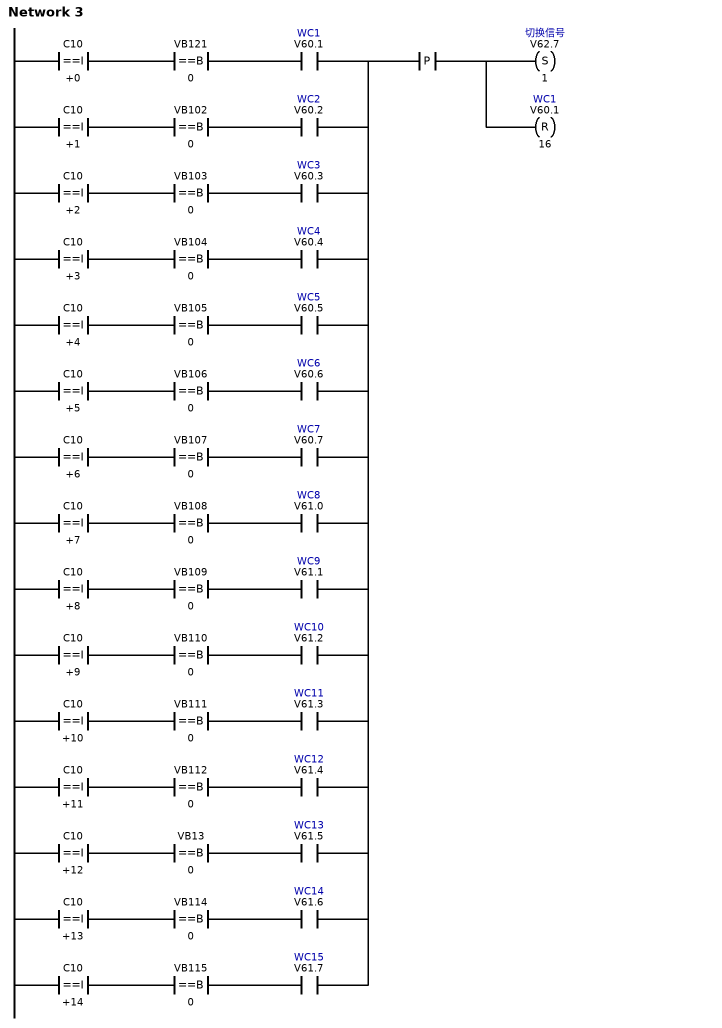
[picture p120: SBR53 networks 3-3]
Network 3
LDW=   C10, +0
AB=    VB121, 0
A      WC1:V60.1
LDW=   C10, +1
AB=    VB102, 0
A      WC2:V60.2
OLD
LDW=   C10, +2
AB=    VB103, 0
A      WC3:V60.3
OLD
LDW=   C10, +3
AB=    VB104, 0
A      WC4:V60.4
OLD
LDW=   C10, +4
AB=    VB105, 0
A      WC5:V60.5
OLD
LDW=   C10, +5
AB=    VB106, 0
A      WC6:V60.6
OLD
LDW=   C10, +6
AB=    VB107, 0
A      WC7:V60.7
OLD
LDW=   C10, +7
AB=    VB108, 0
A      WC8:V61.0
OLD
LDW=   C10, +8
AB=    VB109, 0
A      WC9:V61.1
OLD
LDW=   C10, +9
AB=    VB110, 0
A      WC10:V61.2
OLD
LDW=   C10, +10
AB=    VB111, 0
A      WC11:V61.3
OLD
LDW=   C10, +11
AB=    VB112, 0
A      WC12:V61.4
OLD
LDW=   C10, +12
AB=    VB13, 0
A      WC13:V61.5
OLD
LDW=   C10, +13
AB=    VB114, 0
A      WC14:V61.6
OLD
LDW=   C10, +14
AB=    VB115, 0
A      WC15:V61.7
OLD
EU
S      切换信号:V62.7, 1
R      WC1:V60.1, 16
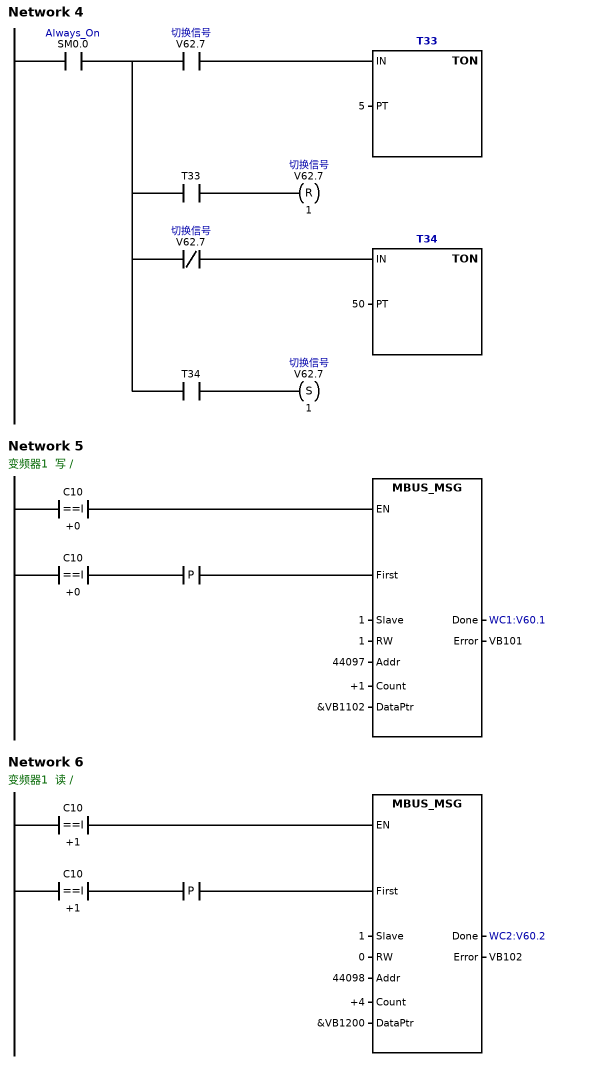
Network 4
LD     Always_On:SM0.0
LPS
A      切换信号:V62.7
TON    T33, 5
LRD
A      T33
R      切换信号:V62.7, 1
LRD
AN     切换信号:V62.7
TON    T34, 50
LPP
A      T34
S      切换信号:V62.7, 1
Network 5
// 变频器1  写
// 
LDW=   C10, +0
=      L60.0
LDW=   C10, +0
EU
=      L63.7
LD     L60.0
CALL   MBUS_MSG:SBR3, L63.7, 1, 1, 44097, +1, &VB1102, WC1:V60.1, VB101
Network 6
// 变频器1  读
// 
LDW=   C10, +1
=      L60.0
LDW=   C10, +1
EU
=      L63.7
LD     L60.0
CALL   MBUS_MSG:SBR3, L63.7, 1, 0, 44098, +4, &VB1200, WC2:V60.2, VB102
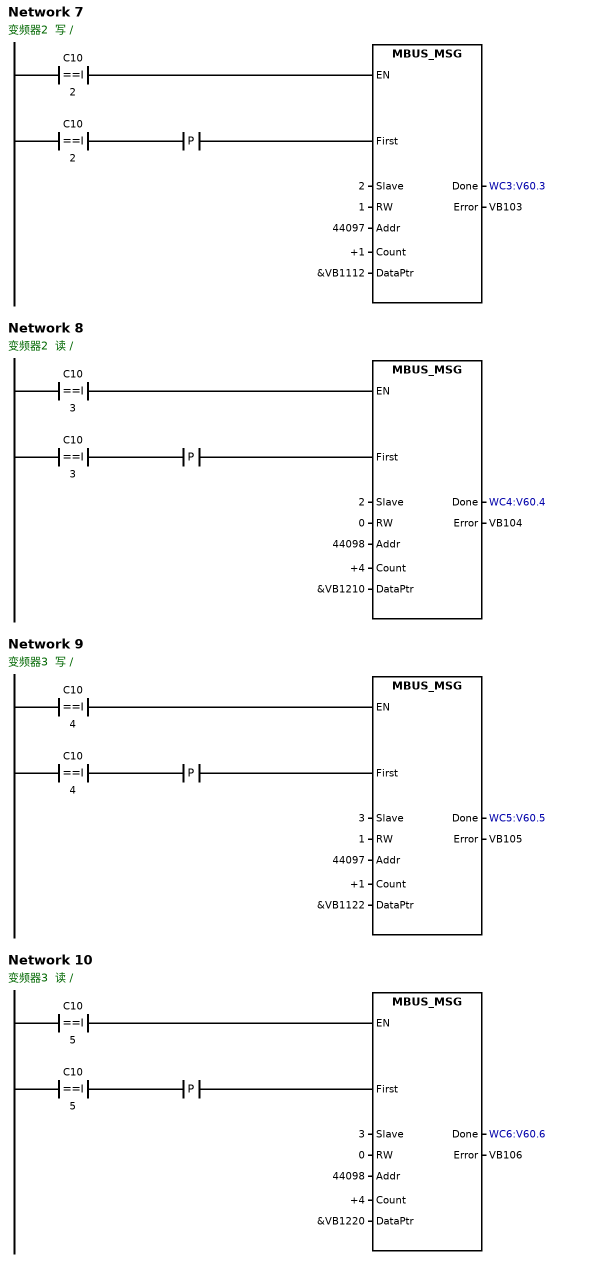
Network 7
// 变频器2  写
// 
LDW=   C10, 2
=      L60.0
LDW=   C10, 2
EU
=      L63.7
LD     L60.0
CALL   MBUS_MSG:SBR3, L63.7, 2, 1, 44097, +1, &VB1112, WC3:V60.3, VB103
Network 8
// 变频器2  读
// 
LDW=   C10, 3
=      L60.0
LDW=   C10, 3
EU
=      L63.7
LD     L60.0
CALL   MBUS_MSG:SBR3, L63.7, 2, 0, 44098, +4, &VB1210, WC4:V60.4, VB104
Network 9
// 变频器3  写
// 
LDW=   C10, 4
=      L60.0
LDW=   C10, 4
EU
=      L63.7
LD     L60.0
CALL   MBUS_MSG:SBR3, L63.7, 3, 1, 44097, +1, &VB1122, WC5:V60.5, VB105
Network 10
// 变频器3  读
// 
LDW=   C10, 5
=      L60.0
LDW=   C10, 5
EU
=      L63.7
LD     L60.0
CALL   MBUS_MSG:SBR3, L63.7, 3, 0, 44098, +4, &VB1220, WC6:V60.6, VB106
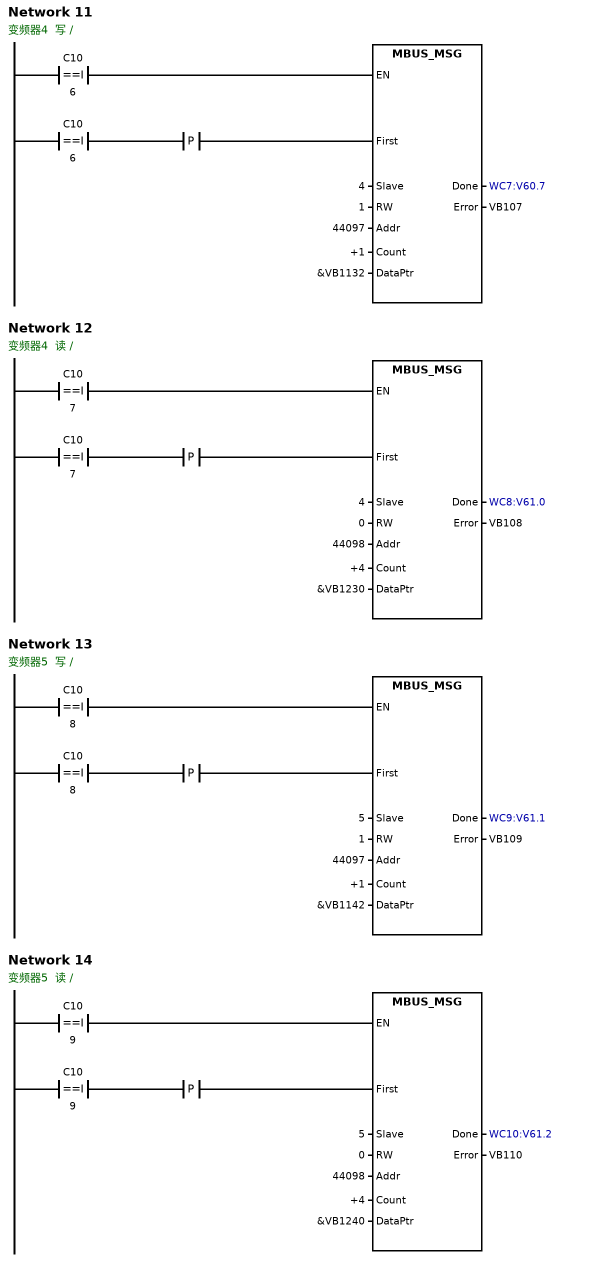
Network 11
// 变频器4  写
// 
LDW=   C10, 6
=      L60.0
LDW=   C10, 6
EU
=      L63.7
LD     L60.0
CALL   MBUS_MSG:SBR3, L63.7, 4, 1, 44097, +1, &VB1132, WC7:V60.7, VB107
Network 12
// 变频器4  读
// 
LDW=   C10, 7
=      L60.0
LDW=   C10, 7
EU
=      L63.7
LD     L60.0
CALL   MBUS_MSG:SBR3, L63.7, 4, 0, 44098, +4, &VB1230, WC8:V61.0, VB108
Network 13
// 变频器5  写
// 
LDW=   C10, 8
=      L60.0
LDW=   C10, 8
EU
=      L63.7
LD     L60.0
CALL   MBUS_MSG:SBR3, L63.7, 5, 1, 44097, +1, &VB1142, WC9:V61.1, VB109
Network 14
// 变频器5  读
// 
LDW=   C10, 9
=      L60.0
LDW=   C10, 9
EU
=      L63.7
LD     L60.0
CALL   MBUS_MSG:SBR3, L63.7, 5, 0, 44098, +4, &VB1240, WC10:V61.2, VB110
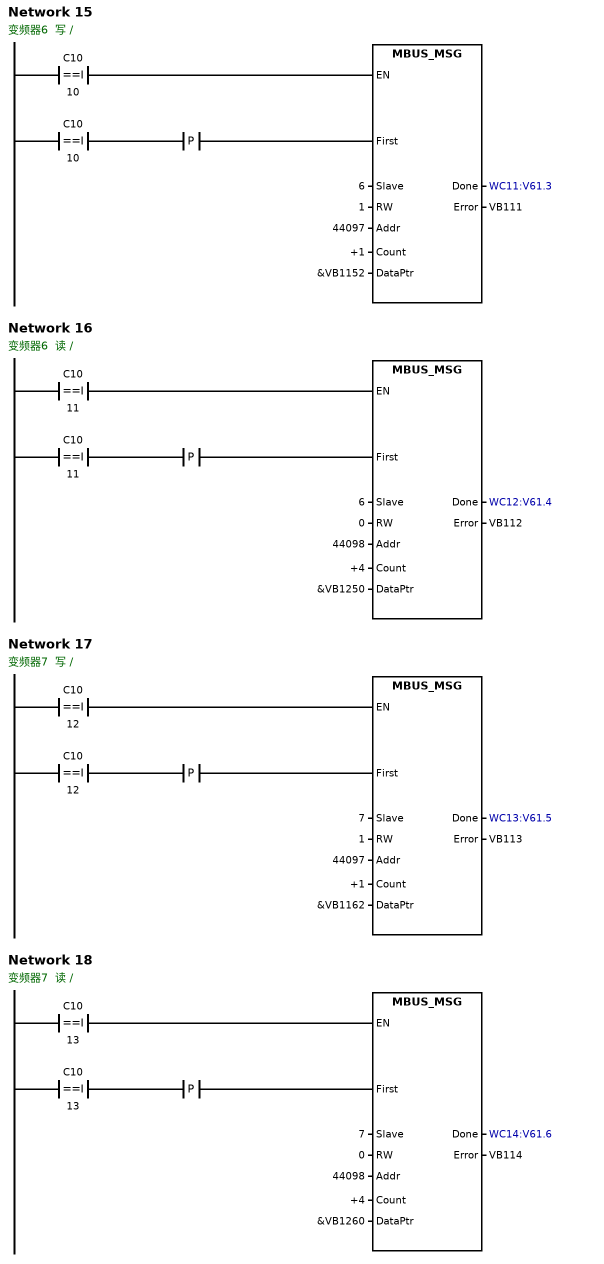
Network 15
// 变频器6  写
// 
LDW=   C10, 10
=      L60.0
LDW=   C10, 10
EU
=      L63.7
LD     L60.0
CALL   MBUS_MSG:SBR3, L63.7, 6, 1, 44097, +1, &VB1152, WC11:V61.3, VB111
Network 16
// 变频器6  读
// 
LDW=   C10, 11
=      L60.0
LDW=   C10, 11
EU
=      L63.7
LD     L60.0
CALL   MBUS_MSG:SBR3, L63.7, 6, 0, 44098, +4, &VB1250, WC12:V61.4, VB112
Network 17
// 变频器7  写
// 
LDW=   C10, 12
=      L60.0
LDW=   C10, 12
EU
=      L63.7
LD     L60.0
CALL   MBUS_MSG:SBR3, L63.7, 7, 1, 44097, +1, &VB1162, WC13:V61.5, VB113
Network 18
// 变频器7  读
// 
LDW=   C10, 13
=      L60.0
LDW=   C10, 13
EU
=      L63.7
LD     L60.0
CALL   MBUS_MSG:SBR3, L63.7, 7, 0, 44098, +4, &VB1260, WC14:V61.6, VB114
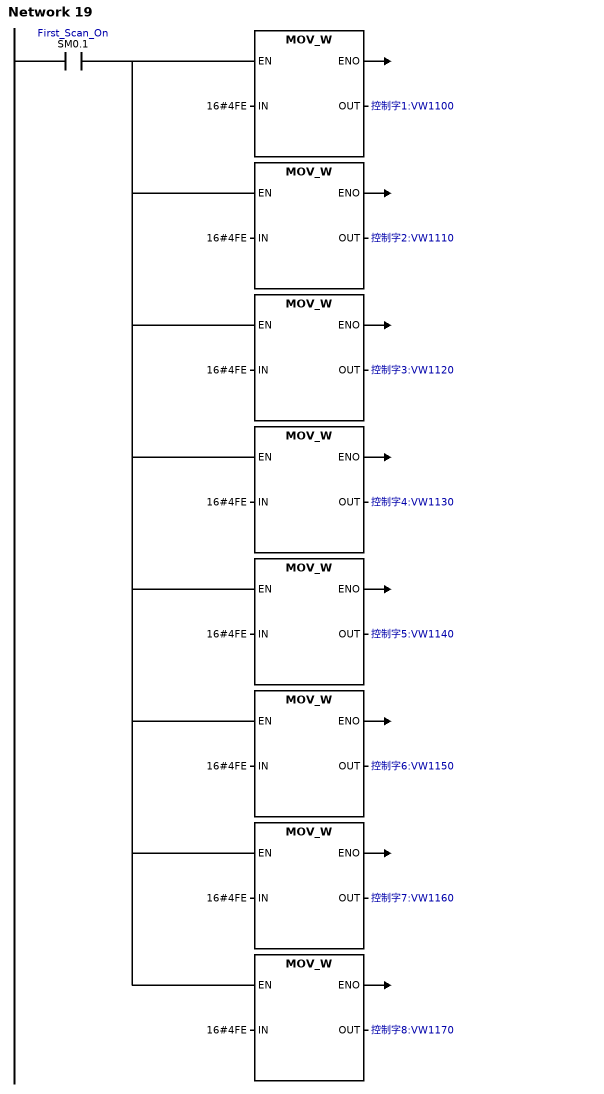
Network 19
LD     First_Scan_On:SM0.1
MOVW   16#4FE, 控制字1:VW1100
MOVW   16#4FE, 控制字2:VW1110
MOVW   16#4FE, 控制字3:VW1120
MOVW   16#4FE, 控制字4:VW1130
MOVW   16#4FE, 控制字5:VW1140
MOVW   16#4FE, 控制字6:VW1150
MOVW   16#4FE, 控制字7:VW1160
MOVW   16#4FE, 控制字8:VW1170
END_SUBROUTINE_BLOCK

SUBROUTINE_BLOCK MODBUS_3610:SBR54
TITLE=
BEGIN
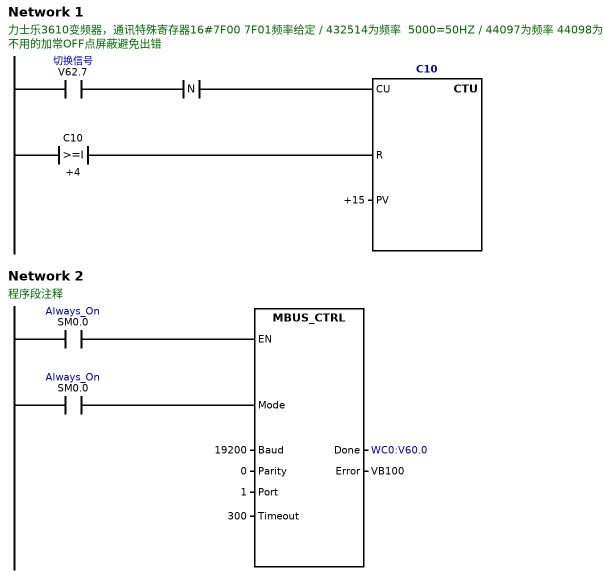
Network 1
// 力士乐3610变频器，通讯特殊寄存器16#7F00 7F01频率给定
// 432514为频率  5000=50HZ
// 44097为频率 44098为电流  通常为2位小数点 1 2
// 波特率19200 无校验
// 16#81  启动 16#88 停止
// 不用的加常OFF点屏蔽避免出错
LD     切换信号:V62.7
ED
LDW>=  C10, +4
CTU    C10, +15
Network 2
// 程序段注释
LD     Always_On:SM0.0
=      L60.0
LD     Always_On:SM0.0
=      L63.7
LD     L60.0
CALL   MBUS_CTRL:SBR2, L63.7, 19200, 0, 1, 300, WC0:V60.0, VB100
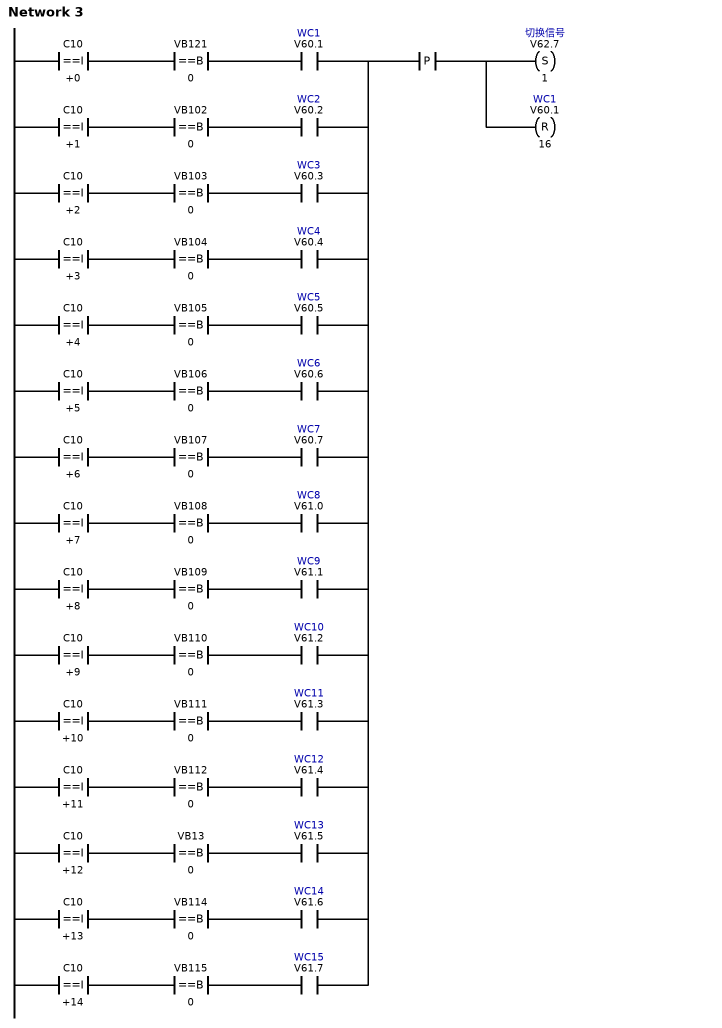
Network 3
LDW=   C10, +0
AB=    VB121, 0
A      WC1:V60.1
LDW=   C10, +1
AB=    VB102, 0
A      WC2:V60.2
OLD
LDW=   C10, +2
AB=    VB103, 0
A      WC3:V60.3
OLD
LDW=   C10, +3
AB=    VB104, 0
A      WC4:V60.4
OLD
LDW=   C10, +4
AB=    VB105, 0
A      WC5:V60.5
OLD
LDW=   C10, +5
AB=    VB106, 0
A      WC6:V60.6
OLD
LDW=   C10, +6
AB=    VB107, 0
A      WC7:V60.7
OLD
LDW=   C10, +7
AB=    VB108, 0
A      WC8:V61.0
OLD
LDW=   C10, +8
AB=    VB109, 0
A      WC9:V61.1
OLD
LDW=   C10, +9
AB=    VB110, 0
A      WC10:V61.2
OLD
LDW=   C10, +10
AB=    VB111, 0
A      WC11:V61.3
OLD
LDW=   C10, +11
AB=    VB112, 0
A      WC12:V61.4
OLD
LDW=   C10, +12
AB=    VB13, 0
A      WC13:V61.5
OLD
LDW=   C10, +13
AB=    VB114, 0
A      WC14:V61.6
OLD
LDW=   C10, +14
AB=    VB115, 0
A      WC15:V61.7
OLD
EU
S      切换信号:V62.7, 1
R      WC1:V60.1, 16
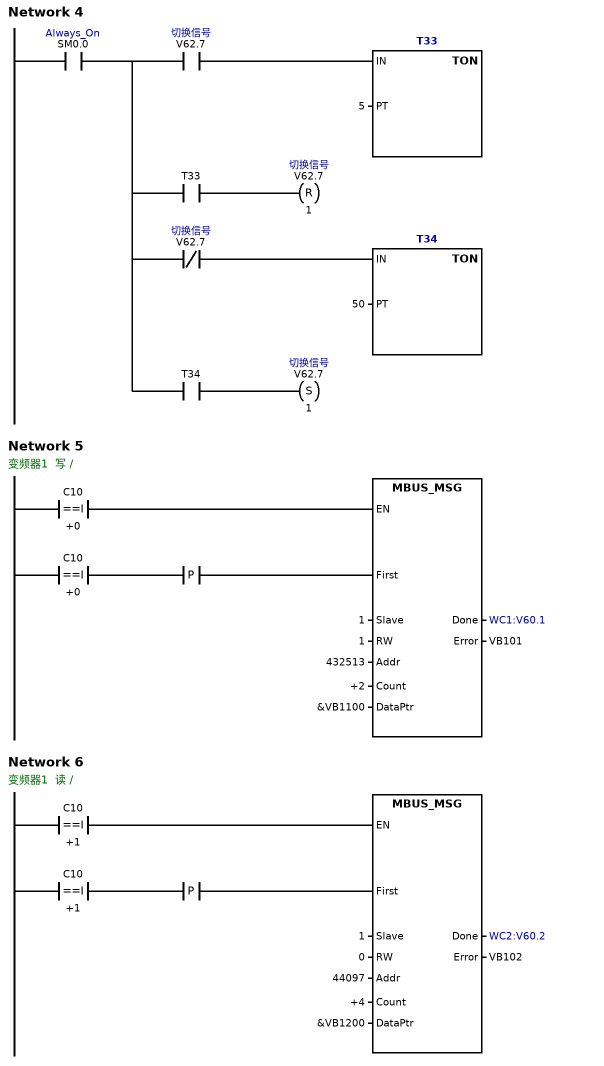
Network 4
LD     Always_On:SM0.0
LPS
A      切换信号:V62.7
TON    T33, 5
LRD
A      T33
R      切换信号:V62.7, 1
LRD
AN     切换信号:V62.7
TON    T34, 50
LPP
A      T34
S      切换信号:V62.7, 1
Network 5
// 变频器1  写
// 
LDW=   C10, +0
=      L60.0
LDW=   C10, +0
EU
=      L63.7
LD     L60.0
CALL   MBUS_MSG:SBR3, L63.7, 1, 1, 432513, +2, &VB1100, WC1:V60.1, VB101
Network 6
// 变频器1  读
// 
LDW=   C10, +1
=      L60.0
LDW=   C10, +1
EU
=      L63.7
LD     L60.0
CALL   MBUS_MSG:SBR3, L63.7, 1, 0, 44097, +4, &VB1200, WC2:V60.2, VB102
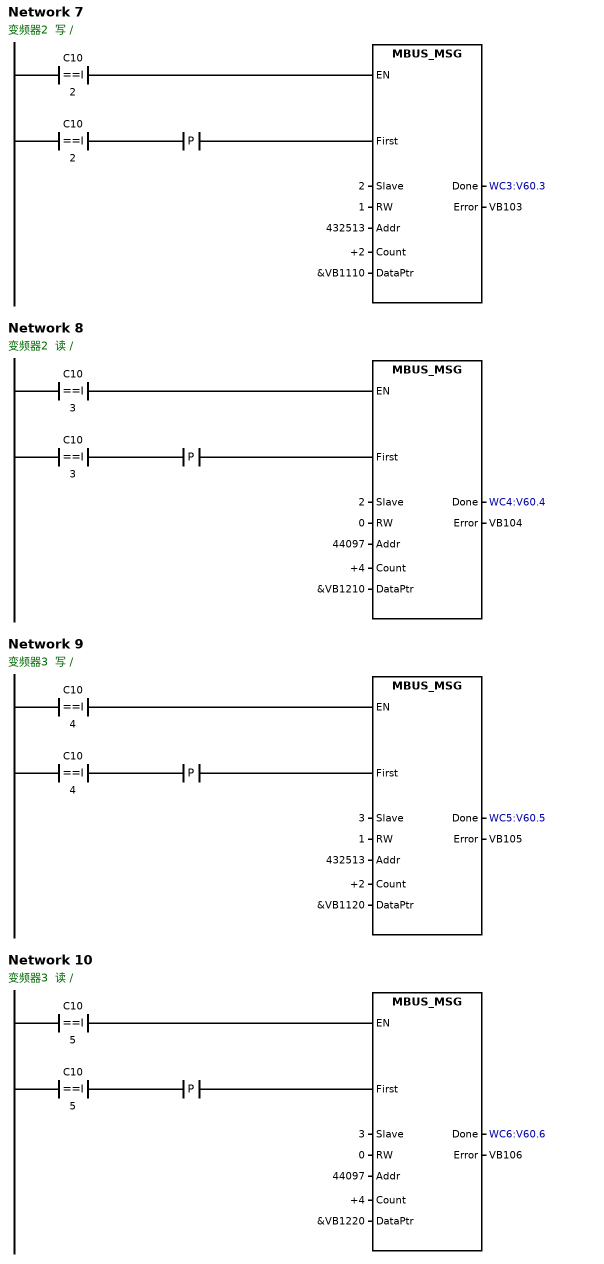
Network 7
// 变频器2  写
// 
LDW=   C10, 2
=      L60.0
LDW=   C10, 2
EU
=      L63.7
LD     L60.0
CALL   MBUS_MSG:SBR3, L63.7, 2, 1, 432513, +2, &VB1110, WC3:V60.3, VB103
Network 8
// 变频器2  读
// 
LDW=   C10, 3
=      L60.0
LDW=   C10, 3
EU
=      L63.7
LD     L60.0
CALL   MBUS_MSG:SBR3, L63.7, 2, 0, 44097, +4, &VB1210, WC4:V60.4, VB104
Network 9
// 变频器3  写
// 
LDW=   C10, 4
=      L60.0
LDW=   C10, 4
EU
=      L63.7
LD     L60.0
CALL   MBUS_MSG:SBR3, L63.7, 3, 1, 432513, +2, &VB1120, WC5:V60.5, VB105
Network 10
// 变频器3  读
// 
LDW=   C10, 5
=      L60.0
LDW=   C10, 5
EU
=      L63.7
LD     L60.0
CALL   MBUS_MSG:SBR3, L63.7, 3, 0, 44097, +4, &VB1220, WC6:V60.6, VB106
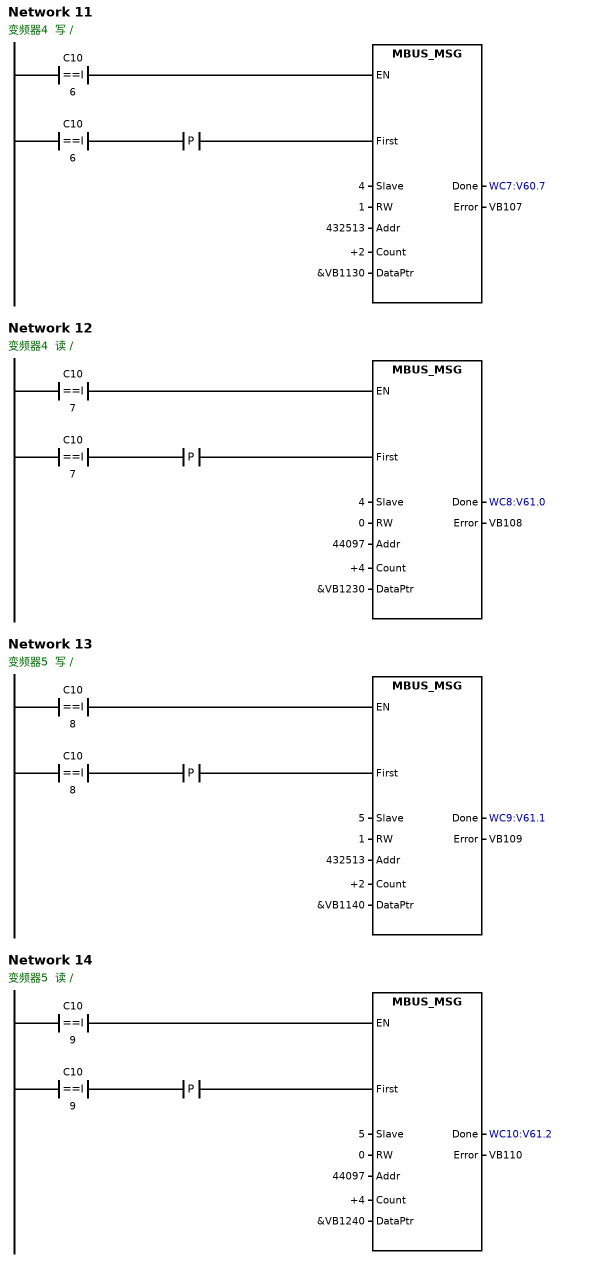
Network 11
// 变频器4  写
// 
LDW=   C10, 6
=      L60.0
LDW=   C10, 6
EU
=      L63.7
LD     L60.0
CALL   MBUS_MSG:SBR3, L63.7, 4, 1, 432513, +2, &VB1130, WC7:V60.7, VB107
Network 12
// 变频器4  读
// 
LDW=   C10, 7
=      L60.0
LDW=   C10, 7
EU
=      L63.7
LD     L60.0
CALL   MBUS_MSG:SBR3, L63.7, 4, 0, 44097, +4, &VB1230, WC8:V61.0, VB108
Network 13
// 变频器5  写
// 
LDW=   C10, 8
=      L60.0
LDW=   C10, 8
EU
=      L63.7
LD     L60.0
CALL   MBUS_MSG:SBR3, L63.7, 5, 1, 432513, +2, &VB1140, WC9:V61.1, VB109
Network 14
// 变频器5  读
// 
LDW=   C10, 9
=      L60.0
LDW=   C10, 9
EU
=      L63.7
LD     L60.0
CALL   MBUS_MSG:SBR3, L63.7, 5, 0, 44097, +4, &VB1240, WC10:V61.2, VB110
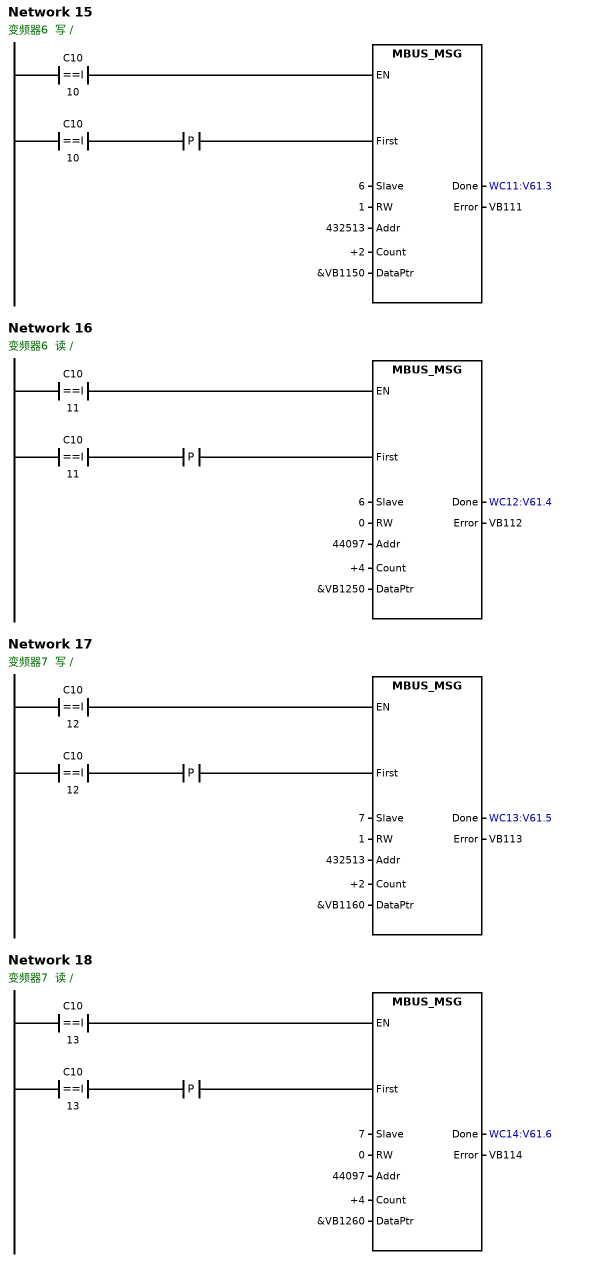
Network 15
// 变频器6  写
// 
LDW=   C10, 10
=      L60.0
LDW=   C10, 10
EU
=      L63.7
LD     L60.0
CALL   MBUS_MSG:SBR3, L63.7, 6, 1, 432513, +2, &VB1150, WC11:V61.3, VB111
Network 16
// 变频器6  读
// 
LDW=   C10, 11
=      L60.0
LDW=   C10, 11
EU
=      L63.7
LD     L60.0
CALL   MBUS_MSG:SBR3, L63.7, 6, 0, 44097, +4, &VB1250, WC12:V61.4, VB112
Network 17
// 变频器7  写
// 
LDW=   C10, 12
=      L60.0
LDW=   C10, 12
EU
=      L63.7
LD     L60.0
CALL   MBUS_MSG:SBR3, L63.7, 7, 1, 432513, +2, &VB1160, WC13:V61.5, VB113
Network 18
// 变频器7  读
// 
LDW=   C10, 13
=      L60.0
LDW=   C10, 13
EU
=      L63.7
LD     L60.0
CALL   MBUS_MSG:SBR3, L63.7, 7, 0, 44097, +4, &VB1260, WC14:V61.6, VB114
END_SUBROUTINE_BLOCK

SUBROUTINE_BLOCK MODBUS_ABB:SBR55
TITLE=
BEGIN
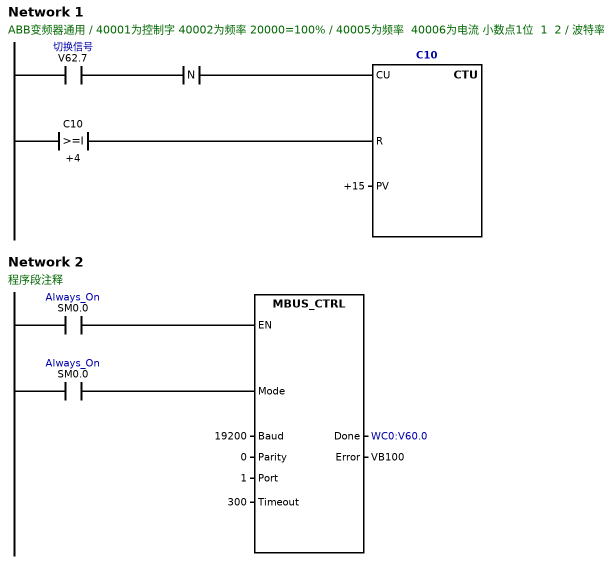
Network 1
// ABB变频器通用
// 40001为控制字 40002为频率 20000=100%
// 40005为频率  40006为电流 小数点1位  1  2
// 波特率19200 无校验
// 16#0477停  16#047F启  16#04F6复位
// 不用的加常OFF点屏蔽避免出错
LD     切换信号:V62.7
ED
LDW>=  C10, +4
CTU    C10, +15
Network 2
// 程序段注释
LD     Always_On:SM0.0
=      L60.0
LD     Always_On:SM0.0
=      L63.7
LD     L60.0
CALL   MBUS_CTRL:SBR2, L63.7, 19200, 0, 1, 300, WC0:V60.0, VB100
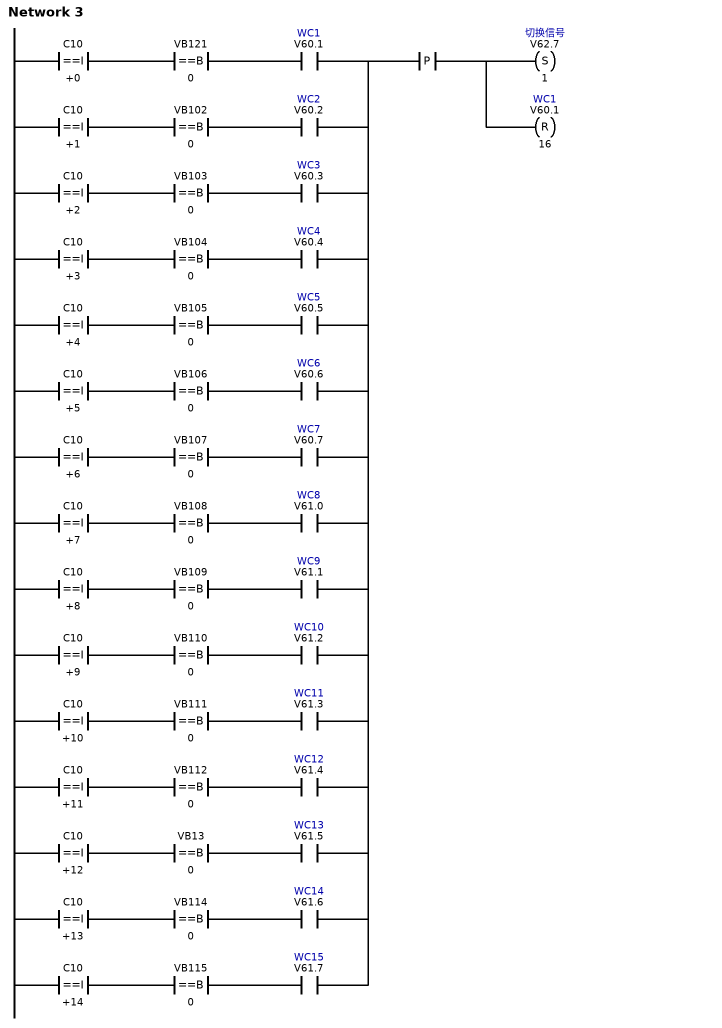
Network 3
LDW=   C10, +0
AB=    VB121, 0
A      WC1:V60.1
LDW=   C10, +1
AB=    VB102, 0
A      WC2:V60.2
OLD
LDW=   C10, +2
AB=    VB103, 0
A      WC3:V60.3
OLD
LDW=   C10, +3
AB=    VB104, 0
A      WC4:V60.4
OLD
LDW=   C10, +4
AB=    VB105, 0
A      WC5:V60.5
OLD
LDW=   C10, +5
AB=    VB106, 0
A      WC6:V60.6
OLD
LDW=   C10, +6
AB=    VB107, 0
A      WC7:V60.7
OLD
LDW=   C10, +7
AB=    VB108, 0
A      WC8:V61.0
OLD
LDW=   C10, +8
AB=    VB109, 0
A      WC9:V61.1
OLD
LDW=   C10, +9
AB=    VB110, 0
A      WC10:V61.2
OLD
LDW=   C10, +10
AB=    VB111, 0
A      WC11:V61.3
OLD
LDW=   C10, +11
AB=    VB112, 0
A      WC12:V61.4
OLD
LDW=   C10, +12
AB=    VB13, 0
A      WC13:V61.5
OLD
LDW=   C10, +13
AB=    VB114, 0
A      WC14:V61.6
OLD
LDW=   C10, +14
AB=    VB115, 0
A      WC15:V61.7
OLD
EU
S      切换信号:V62.7, 1
R      WC1:V60.1, 16
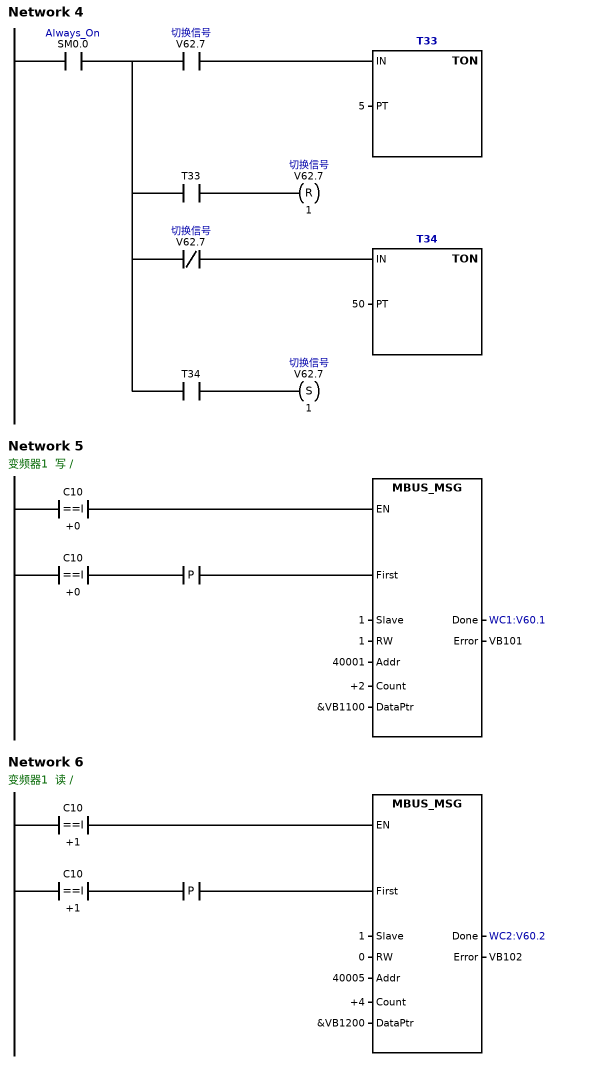
Network 4
LD     Always_On:SM0.0
LPS
A      切换信号:V62.7
TON    T33, 5
LRD
A      T33
R      切换信号:V62.7, 1
LRD
AN     切换信号:V62.7
TON    T34, 50
LPP
A      T34
S      切换信号:V62.7, 1
Network 5
// 变频器1  写
// 
LDW=   C10, +0
=      L60.0
LDW=   C10, +0
EU
=      L63.7
LD     L60.0
CALL   MBUS_MSG:SBR3, L63.7, 1, 1, 40001, +2, &VB1100, WC1:V60.1, VB101
Network 6
// 变频器1  读
// 
LDW=   C10, +1
=      L60.0
LDW=   C10, +1
EU
=      L63.7
LD     L60.0
CALL   MBUS_MSG:SBR3, L63.7, 1, 0, 40005, +4, &VB1200, WC2:V60.2, VB102
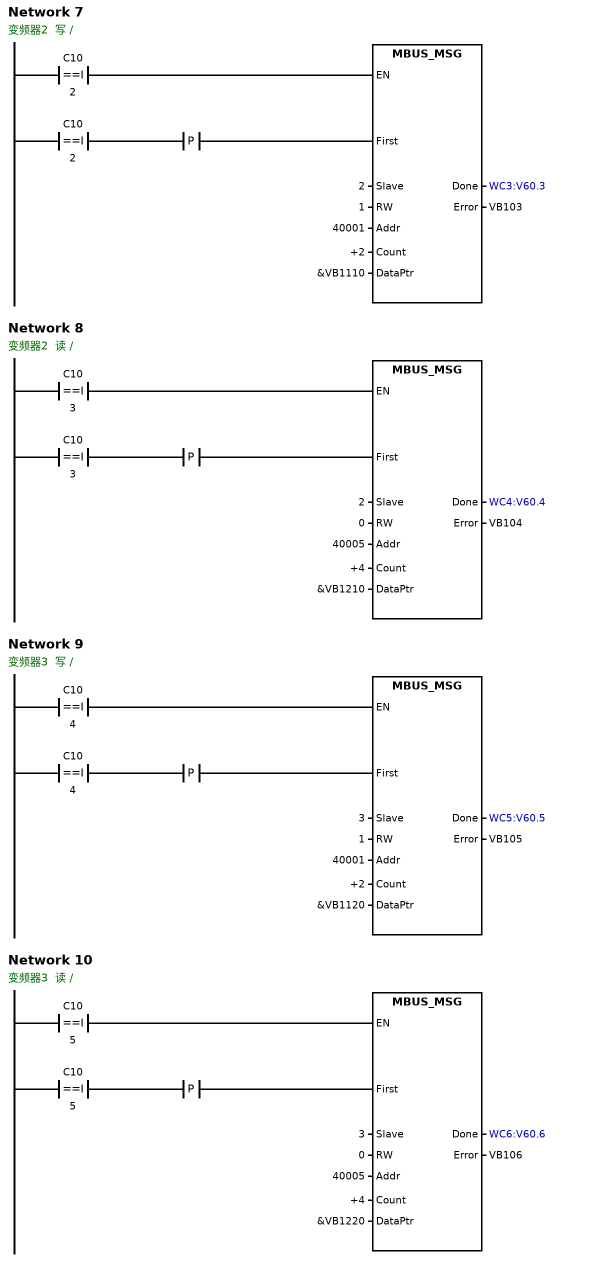
Network 7
// 变频器2  写
// 
LDW=   C10, 2
=      L60.0
LDW=   C10, 2
EU
=      L63.7
LD     L60.0
CALL   MBUS_MSG:SBR3, L63.7, 2, 1, 40001, +2, &VB1110, WC3:V60.3, VB103
Network 8
// 变频器2  读
// 
LDW=   C10, 3
=      L60.0
LDW=   C10, 3
EU
=      L63.7
LD     L60.0
CALL   MBUS_MSG:SBR3, L63.7, 2, 0, 40005, +4, &VB1210, WC4:V60.4, VB104
Network 9
// 变频器3  写
// 
LDW=   C10, 4
=      L60.0
LDW=   C10, 4
EU
=      L63.7
LD     L60.0
CALL   MBUS_MSG:SBR3, L63.7, 3, 1, 40001, +2, &VB1120, WC5:V60.5, VB105
Network 10
// 变频器3  读
// 
LDW=   C10, 5
=      L60.0
LDW=   C10, 5
EU
=      L63.7
LD     L60.0
CALL   MBUS_MSG:SBR3, L63.7, 3, 0, 40005, +4, &VB1220, WC6:V60.6, VB106
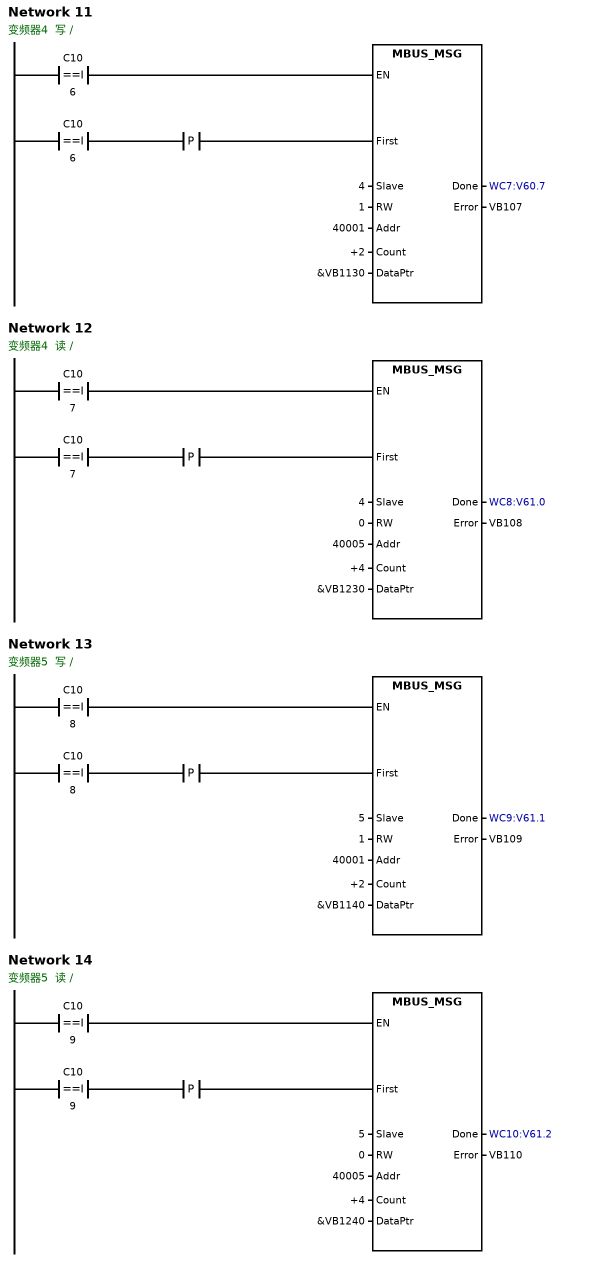
Network 11
// 变频器4  写
// 
LDW=   C10, 6
=      L60.0
LDW=   C10, 6
EU
=      L63.7
LD     L60.0
CALL   MBUS_MSG:SBR3, L63.7, 4, 1, 40001, +2, &VB1130, WC7:V60.7, VB107
Network 12
// 变频器4  读
// 
LDW=   C10, 7
=      L60.0
LDW=   C10, 7
EU
=      L63.7
LD     L60.0
CALL   MBUS_MSG:SBR3, L63.7, 4, 0, 40005, +4, &VB1230, WC8:V61.0, VB108
Network 13
// 变频器5  写
// 
LDW=   C10, 8
=      L60.0
LDW=   C10, 8
EU
=      L63.7
LD     L60.0
CALL   MBUS_MSG:SBR3, L63.7, 5, 1, 40001, +2, &VB1140, WC9:V61.1, VB109
Network 14
// 变频器5  读
// 
LDW=   C10, 9
=      L60.0
LDW=   C10, 9
EU
=      L63.7
LD     L60.0
CALL   MBUS_MSG:SBR3, L63.7, 5, 0, 40005, +4, &VB1240, WC10:V61.2, VB110
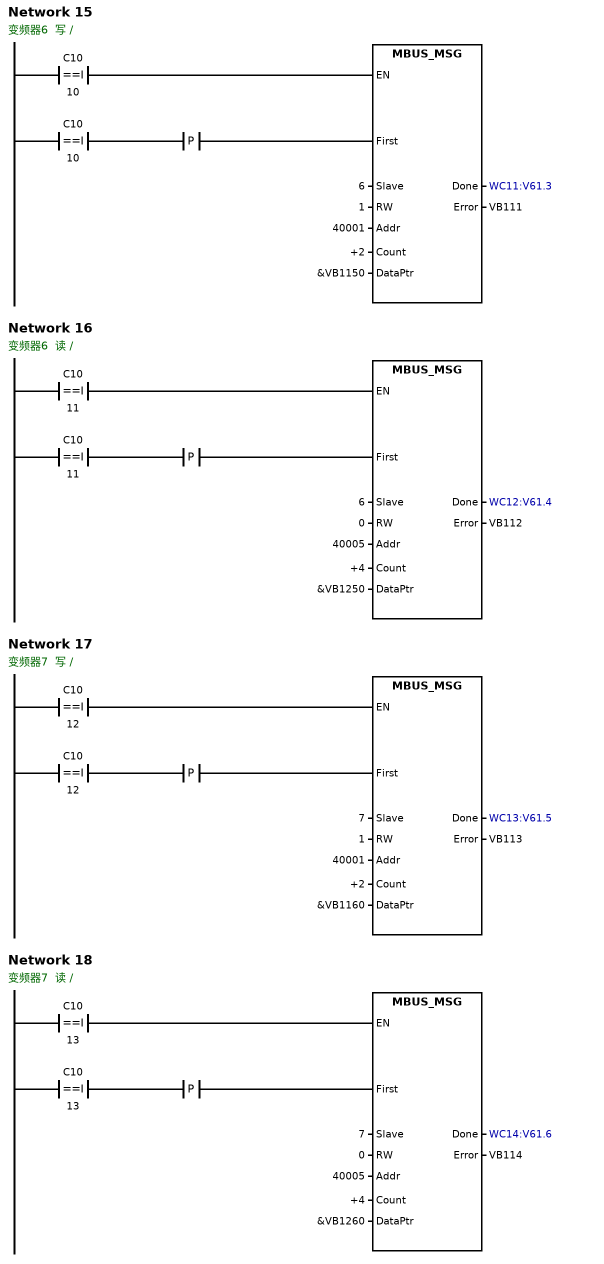
Network 15
// 变频器6  写
// 
LDW=   C10, 10
=      L60.0
LDW=   C10, 10
EU
=      L63.7
LD     L60.0
CALL   MBUS_MSG:SBR3, L63.7, 6, 1, 40001, +2, &VB1150, WC11:V61.3, VB111
Network 16
// 变频器6  读
// 
LDW=   C10, 11
=      L60.0
LDW=   C10, 11
EU
=      L63.7
LD     L60.0
CALL   MBUS_MSG:SBR3, L63.7, 6, 0, 40005, +4, &VB1250, WC12:V61.4, VB112
Network 17
// 变频器7  写
// 
LDW=   C10, 12
=      L60.0
LDW=   C10, 12
EU
=      L63.7
LD     L60.0
CALL   MBUS_MSG:SBR3, L63.7, 7, 1, 40001, +2, &VB1160, WC13:V61.5, VB113
Network 18
// 变频器7  读
// 
LDW=   C10, 13
=      L60.0
LDW=   C10, 13
EU
=      L63.7
LD     L60.0
CALL   MBUS_MSG:SBR3, L63.7, 7, 0, 40005, +4, &VB1260, WC14:V61.6, VB114
END_SUBROUTINE_BLOCK

SUBROUTINE_BLOCK MODBUS三菱:SBR56
TITLE=
BEGIN
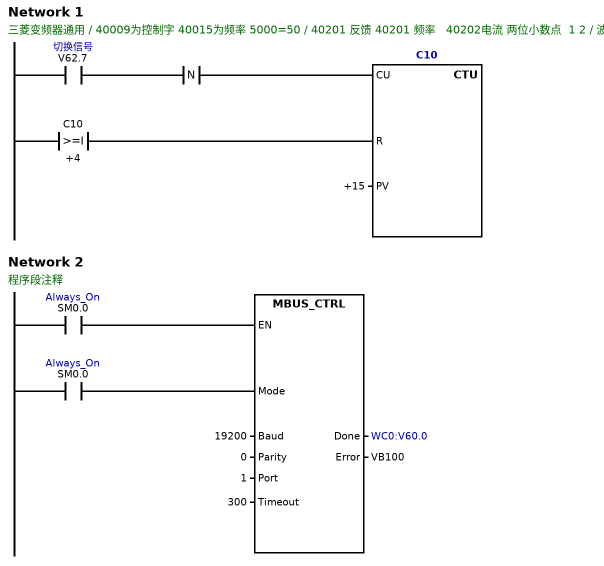
Network 1
// 三菱变频器通用
// 40009为控制字 40015为频率 5000=50
// 40201 反馈 40201 频率   40202电流 两位小数点  1 2
// 波特率19200 无校验
// 0停  1正启 2反启  12复位
// 不用的加常OFF点屏蔽避免出错
LD     切换信号:V62.7
ED
LDW>=  C10, +4
CTU    C10, +15
Network 2
// 程序段注释
LD     Always_On:SM0.0
=      L60.0
LD     Always_On:SM0.0
=      L63.7
LD     L60.0
CALL   MBUS_CTRL:SBR2, L63.7, 19200, 0, 1, 300, WC0:V60.0, VB100
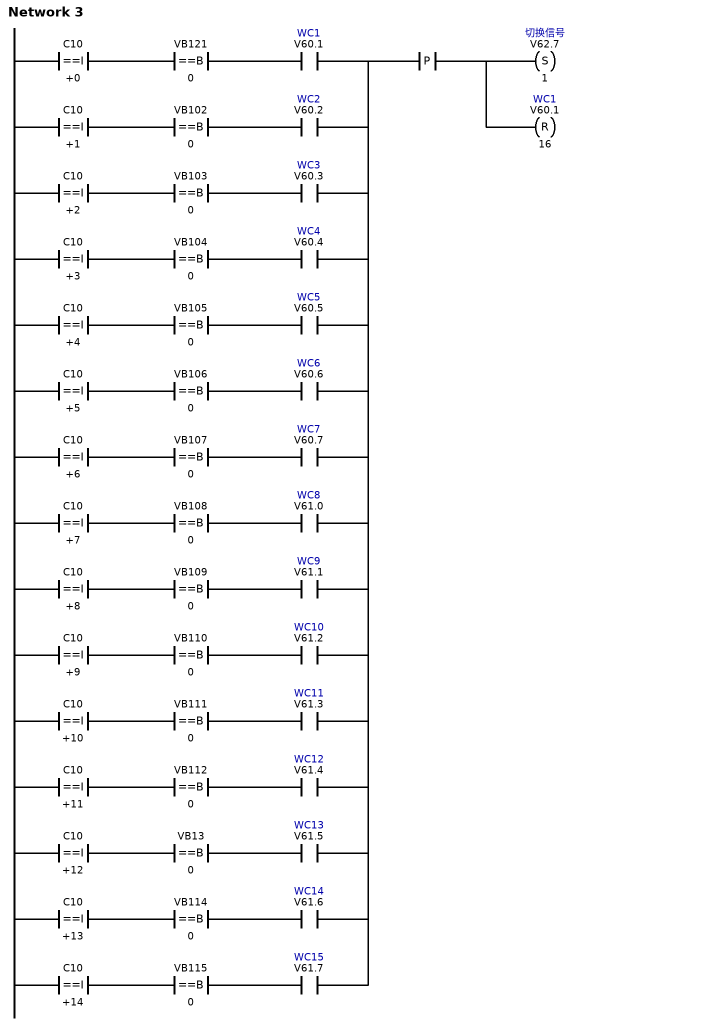
Network 3
LDW=   C10, +0
AB=    VB121, 0
A      WC1:V60.1
LDW=   C10, +1
AB=    VB102, 0
A      WC2:V60.2
OLD
LDW=   C10, +2
AB=    VB103, 0
A      WC3:V60.3
OLD
LDW=   C10, +3
AB=    VB104, 0
A      WC4:V60.4
OLD
LDW=   C10, +4
AB=    VB105, 0
A      WC5:V60.5
OLD
LDW=   C10, +5
AB=    VB106, 0
A      WC6:V60.6
OLD
LDW=   C10, +6
AB=    VB107, 0
A      WC7:V60.7
OLD
LDW=   C10, +7
AB=    VB108, 0
A      WC8:V61.0
OLD
LDW=   C10, +8
AB=    VB109, 0
A      WC9:V61.1
OLD
LDW=   C10, +9
AB=    VB110, 0
A      WC10:V61.2
OLD
LDW=   C10, +10
AB=    VB111, 0
A      WC11:V61.3
OLD
LDW=   C10, +11
AB=    VB112, 0
A      WC12:V61.4
OLD
LDW=   C10, +12
AB=    VB13, 0
A      WC13:V61.5
OLD
LDW=   C10, +13
AB=    VB114, 0
A      WC14:V61.6
OLD
LDW=   C10, +14
AB=    VB115, 0
A      WC15:V61.7
OLD
EU
S      切换信号:V62.7, 1
R      WC1:V60.1, 16
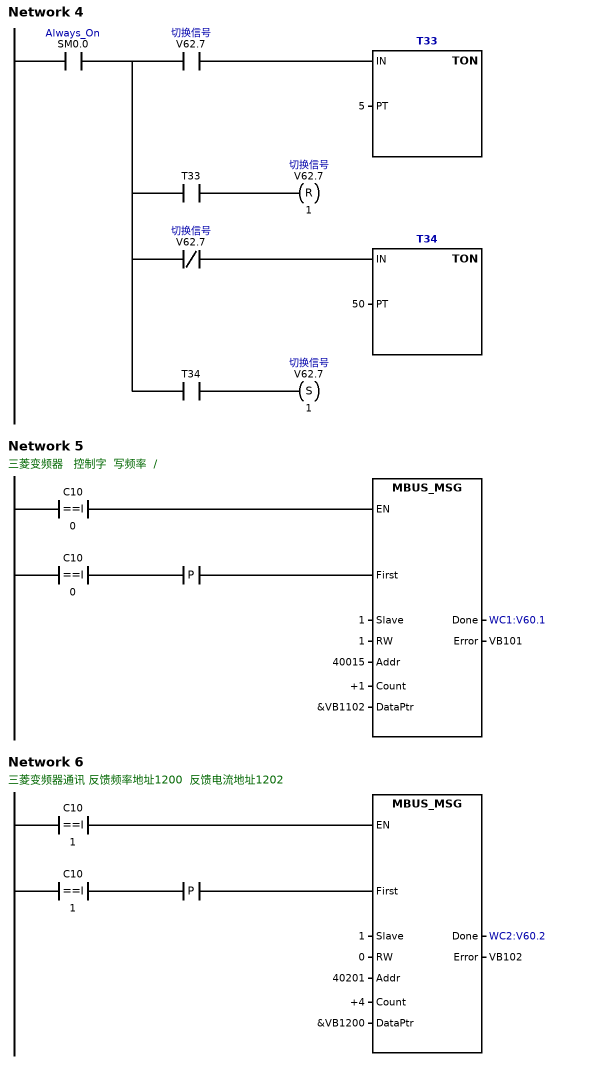
Network 4
LD     Always_On:SM0.0
LPS
A      切换信号:V62.7
TON    T33, 5
LRD
A      T33
R      切换信号:V62.7, 1
LRD
AN     切换信号:V62.7
TON    T34, 50
LPP
A      T34
S      切换信号:V62.7, 1
Network 5
// 三菱变频器   控制字  写频率 
// 
LDW=   C10, 0
=      L60.0
LDW=   C10, 0
EU
=      L63.7
LD     L60.0
CALL   MBUS_MSG:SBR3, L63.7, 1, 1, 40015, +1, &VB1102, WC1:V60.1, VB101
Network 6
// 三菱变频器通讯 反馈频率地址1200  反馈电流地址1202  
LDW=   C10, 1
=      L60.0
LDW=   C10, 1
EU
=      L63.7
LD     L60.0
CALL   MBUS_MSG:SBR3, L63.7, 1, 0, 40201, +4, &VB1200, WC2:V60.2, VB102
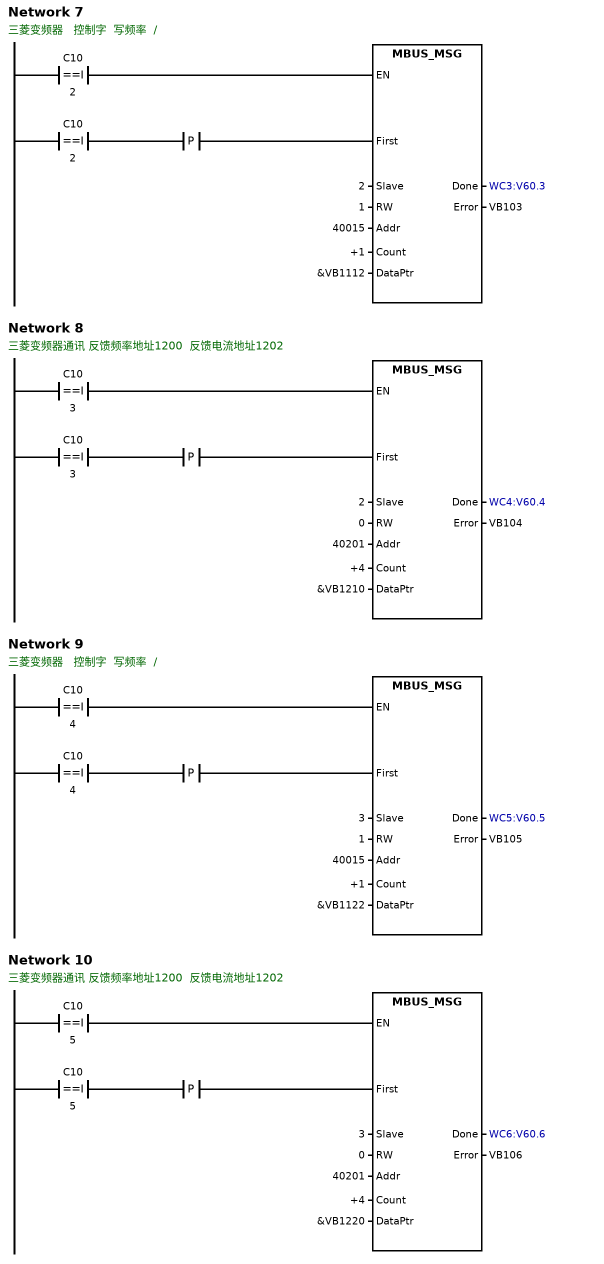
Network 7
// 三菱变频器   控制字  写频率 
// 
LDW=   C10, 2
=      L60.0
LDW=   C10, 2
EU
=      L63.7
LD     L60.0
CALL   MBUS_MSG:SBR3, L63.7, 2, 1, 40015, +1, &VB1112, WC3:V60.3, VB103
Network 8
// 三菱变频器通讯 反馈频率地址1200  反馈电流地址1202  
LDW=   C10, 3
=      L60.0
LDW=   C10, 3
EU
=      L63.7
LD     L60.0
CALL   MBUS_MSG:SBR3, L63.7, 2, 0, 40201, +4, &VB1210, WC4:V60.4, VB104
Network 9
// 三菱变频器   控制字  写频率 
// 
LDW=   C10, 4
=      L60.0
LDW=   C10, 4
EU
=      L63.7
LD     L60.0
CALL   MBUS_MSG:SBR3, L63.7, 3, 1, 40015, +1, &VB1122, WC5:V60.5, VB105
Network 10
// 三菱变频器通讯 反馈频率地址1200  反馈电流地址1202  
LDW=   C10, 5
=      L60.0
LDW=   C10, 5
EU
=      L63.7
LD     L60.0
CALL   MBUS_MSG:SBR3, L63.7, 3, 0, 40201, +4, &VB1220, WC6:V60.6, VB106
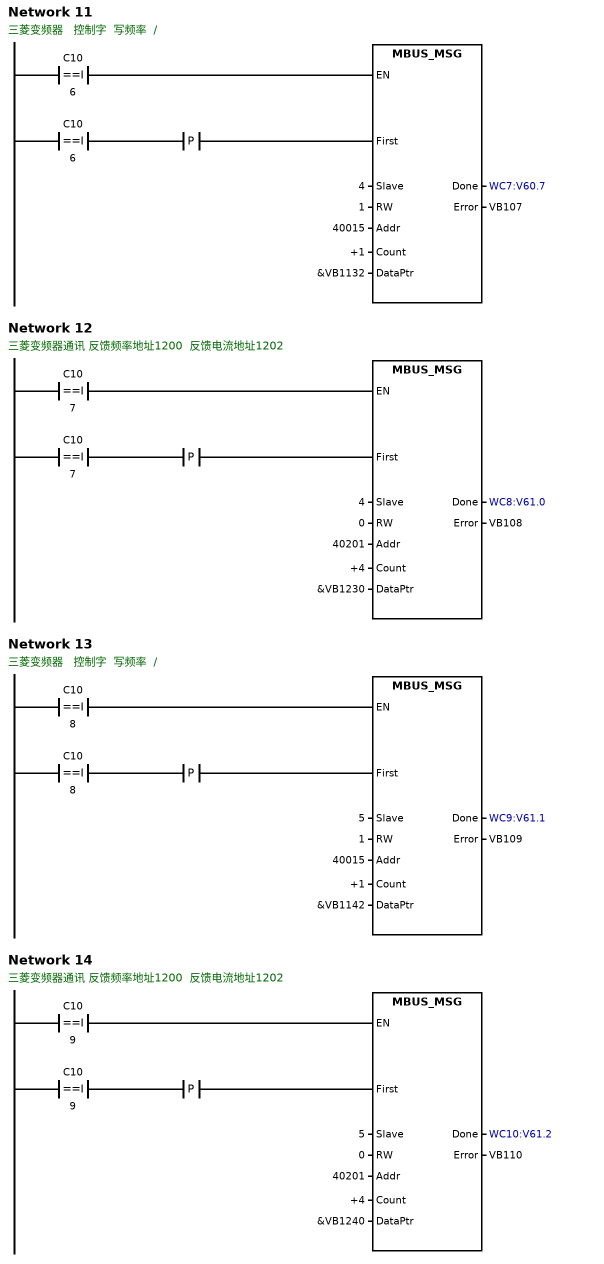
Network 11
// 三菱变频器   控制字  写频率 
// 
LDW=   C10, 6
=      L60.0
LDW=   C10, 6
EU
=      L63.7
LD     L60.0
CALL   MBUS_MSG:SBR3, L63.7, 4, 1, 40015, +1, &VB1132, WC7:V60.7, VB107
Network 12
// 三菱变频器通讯 反馈频率地址1200  反馈电流地址1202  
LDW=   C10, 7
=      L60.0
LDW=   C10, 7
EU
=      L63.7
LD     L60.0
CALL   MBUS_MSG:SBR3, L63.7, 4, 0, 40201, +4, &VB1230, WC8:V61.0, VB108
Network 13
// 三菱变频器   控制字  写频率 
// 
LDW=   C10, 8
=      L60.0
LDW=   C10, 8
EU
=      L63.7
LD     L60.0
CALL   MBUS_MSG:SBR3, L63.7, 5, 1, 40015, +1, &VB1142, WC9:V61.1, VB109
Network 14
// 三菱变频器通讯 反馈频率地址1200  反馈电流地址1202  
LDW=   C10, 9
=      L60.0
LDW=   C10, 9
EU
=      L63.7
LD     L60.0
CALL   MBUS_MSG:SBR3, L63.7, 5, 0, 40201, +4, &VB1240, WC10:V61.2, VB110
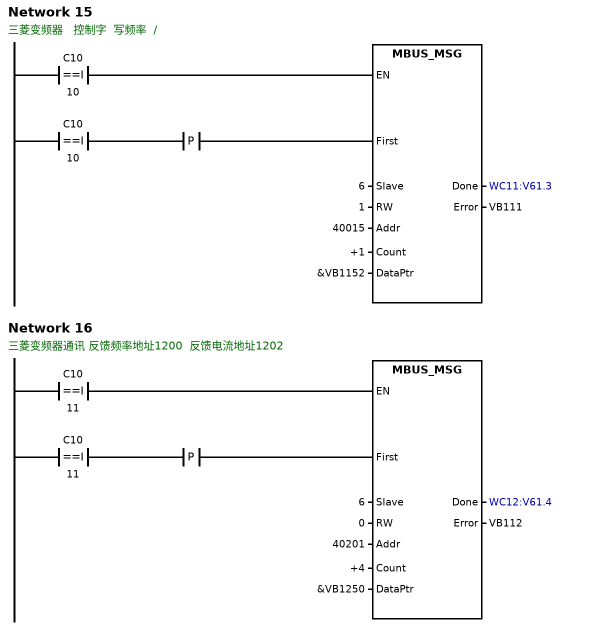
Network 15
// 三菱变频器   控制字  写频率 
// 
LDW=   C10, 10
=      L60.0
LDW=   C10, 10
EU
=      L63.7
LD     L60.0
CALL   MBUS_MSG:SBR3, L63.7, 6, 1, 40015, +1, &VB1152, WC11:V61.3, VB111
Network 16
// 三菱变频器通讯 反馈频率地址1200  反馈电流地址1202  
LDW=   C10, 11
=      L60.0
LDW=   C10, 11
EU
=      L63.7
LD     L60.0
CALL   MBUS_MSG:SBR3, L63.7, 6, 0, 40201, +4, &VB1250, WC12:V61.4, VB112
END_SUBROUTINE_BLOCK

SUBROUTINE_BLOCK MODBUS_电表:SBR58
TITLE=
BEGIN
